(* PLC project PLC, Beckhoff Automation GmbH TwinCAT PLC Control 3.5.21.60 *)
(* stored: creationDateTime 2026-08-05T00:25:24.1454129, modificationDateTime 2026-08-05T00:25:24.1454129 *)

FUNCTION FC_ConcatAll : STRING
VAR_INPUT
	asConcattables					:	ARRAY[0..100] OF STRING;
END_VAR
VAR
	i								:	INT;
	sActual							:	STRING;
	//bStart							:	BOOL := TRUE;
END_VAR

            FOR i := 0 TO 100 BY 1 DO
	IF asConcattables[i] <> '' THEN
		sActual := CONCAT(STR1 := sActual , STR2 := asConcattables[i]);
	END_IF
END_FOR

FC_ConcatAll := sActual;

          
END_FUNCTION

FUNCTION FUN_Build_String_5 : String(255)
VAR_INPUT
	sString_1			:STRING(255);
	sString_2			:STRING(255);
	sString_3			:STRING(255);
	sString_4			:STRING(255);
	sString_5			:STRING(255);
END_VAR
VAR
END_VAR

            IF sString_1 <> ''
	AND sString_2 <>'' 	AND sString_3 <>'' 	AND sString_4 <>'' 	AND sString_5 <>'' THEN
	
	FUN_Build_String_5:=concat(sString_1,concat(sString_2,concat(sString_3,concat(sString_4,sString_5))));
	
ELSIF sString_1 <> ''
	AND sString_2 <>'' 	AND sString_3 <>'' 	AND sString_4 <>'' THEN
	
	FUN_Build_String_5:=concat(sString_1,concat(sString_2,concat(sString_3,sString_4)));
ELSIF sString_1 <> ''
	AND sString_2 <>'' 	AND sString_3 <>'' THEN
	
	FUN_Build_String_5:=concat(sString_1,concat(sString_2,sString_3));
ELSIF sString_1 <> ''AND sString_2 <>'' THEN
	
	FUN_Build_String_5:=concat(sString_1,sString_2);
ELSE
	FUN_Build_String_5:='';
END_IF
          
END_FUNCTION

FUNCTION FUN_Build_String_10 : String(255)
VAR_INPUT
	sString_1			:STRING(255);
	sString_2			:STRING(255);
	sString_3			:STRING(255);
	sString_4			:STRING(255);
	sString_5			:STRING(255);
	sString_6			:STRING(255);
	sString_7			:STRING(255);
	sString_8			:STRING(255);
	sString_9			:STRING(255);
	sString_10			:STRING(255);
END_VAR
VAR
END_VAR

            IF sString_1 <> ''
	AND sString_2 <>'' 	AND sString_3 <>'' 	AND sString_4 <>'' 	AND sString_5 <>'' 	AND sString_6 <>''	AND sString_7 <>''	AND sString_8 <>''
	AND sString_9 <>''	AND sString_10 <>''	 THEN
	
	FUN_Build_String_10:=concat(sString_1,concat(sString_2,concat(sString_3,concat(sString_4,concat
					(sString_5,concat(sString_6,concat(sString_7,concat(sString_8,concat(sString_9,sString_10)))))))));	
ELSIF sString_1 <> ''
	AND sString_2 <>'' 	AND sString_3 <>'' 	AND sString_4 <>'' 	AND sString_5 <>'' 	AND sString_6 <>''	AND sString_7 <>''	AND sString_8 <>''
	AND sString_9 <>'' THEN
	
	FUN_Build_String_10:=concat(sString_1,concat(sString_2,concat(sString_3,concat(sString_4,concat
					(sString_5,concat(sString_6,concat(sString_7,concat(sString_8,sString_9))))))));	
ELSIF sString_1 <> ''
	AND sString_2 <>'' 	AND sString_3 <>'' 	AND sString_4 <>'' 	AND sString_5 <>'' 	AND sString_6 <>''	AND sString_7 <>''	AND sString_8 <>'' THEN
	
	FUN_Build_String_10:=concat(sString_1,concat(sString_2,concat(sString_3,concat(sString_4,concat
					(sString_5,concat(sString_6,concat(sString_7,sString_8)))))));
ELSIF sString_1 <> ''
	AND sString_2 <>'' 	AND sString_3 <>'' 	AND sString_4 <>'' 	AND sString_5 <>'' 	AND sString_6 <>''	AND sString_7 <>'' THEN
	
	FUN_Build_String_10:=concat(sString_1,concat(sString_2,concat(sString_3,concat(sString_4,concat
					(sString_5,concat(sString_6,sString_7))))));
ELSIF sString_1 <> ''
	AND sString_2 <>'' 	AND sString_3 <>'' 	AND sString_4 <>'' 	AND sString_5 <>'' 	AND sString_6 <>'' THEN
	
	FUN_Build_String_10:=concat(sString_1,concat(sString_2,concat(sString_3,concat(sString_4,concat
					(sString_5,sString_6)))));
ELSIF sString_1 <> ''
	AND sString_2 <>'' 	AND sString_3 <>'' 	AND sString_4 <>'' 	AND sString_5 <>'' THEN
	
	FUN_Build_String_10:=concat(sString_1,concat(sString_2,concat(sString_3,concat(sString_4,sString_5))));
	
ELSIF sString_1 <> ''
	AND sString_2 <>'' 	AND sString_3 <>'' 	AND sString_4 <>'' THEN
	
	FUN_Build_String_10:=concat(sString_1,concat(sString_2,concat(sString_3,sString_4)));
ELSIF sString_1 <> ''
	AND sString_2 <>'' 	AND sString_3 <>'' THEN
	
	FUN_Build_String_10:=concat(sString_1,concat(sString_2,sString_3));
ELSIF sString_1 <> ''AND sString_2 <>'' THEN
	
	FUN_Build_String_10:=concat(sString_1,sString_2);
ELSE
	FUN_Build_String_10:='';
END_IF
          
END_FUNCTION

FUNCTION FUN_Build_String_20 : String(255)
VAR_INPUT
	sString_1			:STRING(255);
	sString_2			:STRING(255);
	sString_3			:STRING(255);
	sString_4			:STRING(255);
	sString_5			:STRING(255);
	sString_6			:STRING(255);
	sString_7			:STRING(255);
	sString_8			:STRING(255);
	sString_9			:STRING(255);
	sString_10			:STRING(255);
	sString_11			:STRING(255);
	sString_12			:STRING(255);
	sString_13			:STRING(255);
	sString_14			:STRING(255);
	sString_15			:STRING(255);
	sString_16			:STRING(255);
	sString_17			:STRING(255);
	sString_18			:STRING(255);
	sString_19			:STRING(255);
	sString_20			:STRING(255);
END_VAR
VAR
END_VAR

            IF sString_1 <> ''
	AND sString_2 <>'' 	AND sString_3 <>'' 	AND sString_4 <>'' 	AND sString_5 <>'' 	AND sString_6 <>''	AND sString_7 <>''	AND sString_8 <>''
	AND sString_9 <>''	AND sString_10 <>''	AND sString_11 <>''	AND sString_12 <>'' AND sString_13 <>''	AND sString_14 <>''	AND sString_15 <>''
	AND sString_16 <>''	AND sString_17 <>''	AND sString_18 <>''	AND sString_19 <>''	AND sString_20 <>'' THEN
	
	FUN_Build_String_20:=concat(sString_1,concat(sString_2,concat(sString_3,concat(sString_4,concat
					(sString_5,concat(sString_6,concat(sString_7,concat(sString_8,concat(sString_9,
						concat(sString_10,concat(sString_11,concat(sString_12,concat(sString_13,concat(sString_14,
							concat(sString_15,concat(sString_16,concat(sString_17,concat(sString_18,concat(sString_19,sString_20)))))))))))))))))));
ELSIF sString_1 <> ''
	AND sString_2 <>'' 	AND sString_3 <>'' 	AND sString_4 <>'' 	AND sString_5 <>'' 	AND sString_6 <>''	AND sString_7 <>''	AND sString_8 <>''
	AND sString_9 <>''	AND sString_10 <>''	AND sString_11 <>''	AND sString_12 <>'' AND sString_13 <>''	AND sString_14 <>''	AND sString_15 <>''
	AND sString_16 <>''	AND sString_17 <>''	AND sString_18 <>''	AND sString_19 <>''	 THEN
	
	FUN_Build_String_20:=concat(sString_1,concat(sString_2,concat(sString_3,concat(sString_4,concat
					(sString_5,concat(sString_6,concat(sString_7,concat(sString_8,concat(sString_9,
						concat(sString_10,concat(sString_11,concat(sString_12,concat(sString_13,concat(sString_14,
							concat(sString_15,concat(sString_16,concat(sString_17,concat(sString_18,sString_19))))))))))))))))));
ELSIF sString_1 <> ''
	AND sString_2 <>'' 	AND sString_3 <>'' 	AND sString_4 <>'' 	AND sString_5 <>'' 	AND sString_6 <>''	AND sString_7 <>''	AND sString_8 <>''
	AND sString_9 <>''	AND sString_10 <>''	AND sString_11 <>''	AND sString_12 <>'' AND sString_13 <>''	AND sString_14 <>''	AND sString_15 <>''
	AND sString_16 <>''	AND sString_17 <>''	AND sString_18 <>'' THEN
	
	FUN_Build_String_20:=concat(sString_1,concat(sString_2,concat(sString_3,concat(sString_4,concat
					(sString_5,concat(sString_6,concat(sString_7,concat(sString_8,concat(sString_9,
						concat(sString_10,concat(sString_11,concat(sString_12,concat(sString_13,concat(sString_14,
							concat(sString_15,concat(sString_16,concat(sString_17,sString_18)))))))))))))))));	
ELSIF sString_1 <> ''
	AND sString_2 <>'' 	AND sString_3 <>'' 	AND sString_4 <>'' 	AND sString_5 <>'' 	AND sString_6 <>''	AND sString_7 <>''	AND sString_8 <>''
	AND sString_9 <>''	AND sString_10 <>''	AND sString_11 <>''	AND sString_12 <>'' AND sString_13 <>''	AND sString_14 <>''	AND sString_15 <>''
	AND sString_16 <>''	AND sString_17 <>'' THEN
	
	FUN_Build_String_20:=concat(sString_1,concat(sString_2,concat(sString_3,concat(sString_4,concat
					(sString_5,concat(sString_6,concat(sString_7,concat(sString_8,concat(sString_9,
						concat(sString_10,concat(sString_11,concat(sString_12,concat(sString_13,concat(sString_14,
							concat(sString_15,concat(sString_16,sString_17))))))))))))))));	
ELSIF sString_1 <> ''
	AND sString_2 <>'' 	AND sString_3 <>'' 	AND sString_4 <>'' 	AND sString_5 <>'' 	AND sString_6 <>''	AND sString_7 <>''	AND sString_8 <>''
	AND sString_9 <>''	AND sString_10 <>''	AND sString_11 <>''	AND sString_12 <>'' AND sString_13 <>''	AND sString_14 <>''	AND sString_15 <>''
	AND sString_16 <>''	THEN
	
	FUN_Build_String_20:=concat(sString_1,concat(sString_2,concat(sString_3,concat(sString_4,concat
					(sString_5,concat(sString_6,concat(sString_7,concat(sString_8,concat(sString_9,
						concat(sString_10,concat(sString_11,concat(sString_12,concat(sString_13,concat(sString_14,
							concat(sString_15,sString_16)))))))))))))));	
ELSIF sString_1 <> ''
	AND sString_2 <>'' 	AND sString_3 <>'' 	AND sString_4 <>'' 	AND sString_5 <>'' 	AND sString_6 <>''	AND sString_7 <>''	AND sString_8 <>''
	AND sString_9 <>''	AND sString_10 <>''	AND sString_11 <>''	AND sString_12 <>'' AND sString_13 <>''	AND sString_14 <>''	AND sString_15 <>''	THEN
	
	FUN_Build_String_20:=concat(sString_1,concat(sString_2,concat(sString_3,concat(sString_4,concat
					(sString_5,concat(sString_6,concat(sString_7,concat(sString_8,concat(sString_9,
						concat(sString_10,concat(sString_11,concat(sString_12,concat(sString_13,concat(sString_14,sString_15))))))))))))));	
ELSIF sString_1 <> ''
	AND sString_2 <>'' 	AND sString_3 <>'' 	AND sString_4 <>'' 	AND sString_5 <>'' 	AND sString_6 <>''	AND sString_7 <>''	AND sString_8 <>''
	AND sString_9 <>''	AND sString_10 <>''	AND sString_11 <>''	AND sString_12 <>'' AND sString_13 <>''	AND sString_14 <>'' THEN
	
	FUN_Build_String_20:=concat(sString_1,concat(sString_2,concat(sString_3,concat(sString_4,concat
					(sString_5,concat(sString_6,concat(sString_7,concat(sString_8,concat(sString_9,
						concat(sString_10,concat(sString_11,concat(sString_12,concat(sString_13,sString_14)))))))))))));	
ELSIF sString_1 <> ''
	AND sString_2 <>'' 	AND sString_3 <>'' 	AND sString_4 <>'' 	AND sString_5 <>'' 	AND sString_6 <>''	AND sString_7 <>''	AND sString_8 <>''
	AND sString_9 <>''	AND sString_10 <>''	AND sString_11 <>''	AND sString_12 <>'' AND sString_13 <>'' THEN
	
	FUN_Build_String_20:=concat(sString_1,concat(sString_2,concat(sString_3,concat(sString_4,concat
					(sString_5,concat(sString_6,concat(sString_7,concat(sString_8,concat(sString_9,
						concat(sString_10,concat(sString_11,concat(sString_12,sString_13))))))))))));	
ELSIF sString_1 <> ''
	AND sString_2 <>'' 	AND sString_3 <>'' 	AND sString_4 <>'' 	AND sString_5 <>'' 	AND sString_6 <>''	AND sString_7 <>''	AND sString_8 <>''
	AND sString_9 <>''	AND sString_10 <>''	AND sString_11 <>''	AND sString_12 <>'' THEN
	
	FUN_Build_String_20:=concat(sString_1,concat(sString_2,concat(sString_3,concat(sString_4,concat
					(sString_5,concat(sString_6,concat(sString_7,concat(sString_8,concat(sString_9,
						concat(sString_10,concat(sString_11,sString_12)))))))))));	
ELSIF sString_1 <> ''
	AND sString_2 <>'' 	AND sString_3 <>'' 	AND sString_4 <>'' 	AND sString_5 <>'' 	AND sString_6 <>''	AND sString_7 <>''	AND sString_8 <>''
	AND sString_9 <>''	AND sString_10 <>''	AND sString_11 <>'' THEN
	
	FUN_Build_String_20:=concat(sString_1,concat(sString_2,concat(sString_3,concat(sString_4,concat
					(sString_5,concat(sString_6,concat(sString_7,concat(sString_8,concat(sString_9,
						concat(sString_10,sString_11))))))))));	
ELSIF sString_1 <> ''
	AND sString_2 <>'' 	AND sString_3 <>'' 	AND sString_4 <>'' 	AND sString_5 <>'' 	AND sString_6 <>''	AND sString_7 <>''	AND sString_8 <>''
	AND sString_9 <>''	AND sString_10 <>''	 THEN
	
	FUN_Build_String_20:=concat(sString_1,concat(sString_2,concat(sString_3,concat(sString_4,concat
					(sString_5,concat(sString_6,concat(sString_7,concat(sString_8,concat(sString_9,sString_10)))))))));	
ELSIF sString_1 <> ''
	AND sString_2 <>'' 	AND sString_3 <>'' 	AND sString_4 <>'' 	AND sString_5 <>'' 	AND sString_6 <>''	AND sString_7 <>''	AND sString_8 <>''
	AND sString_9 <>'' THEN
	
	FUN_Build_String_20:=concat(sString_1,concat(sString_2,concat(sString_3,concat(sString_4,concat
					(sString_5,concat(sString_6,concat(sString_7,concat(sString_8,sString_9))))))));	
ELSIF sString_1 <> ''
	AND sString_2 <>'' 	AND sString_3 <>'' 	AND sString_4 <>'' 	AND sString_5 <>'' 	AND sString_6 <>''	AND sString_7 <>''	AND sString_8 <>'' THEN
	
	FUN_Build_String_20:=concat(sString_1,concat(sString_2,concat(sString_3,concat(sString_4,concat
					(sString_5,concat(sString_6,concat(sString_7,sString_8)))))));
ELSIF sString_1 <> ''
	AND sString_2 <>'' 	AND sString_3 <>'' 	AND sString_4 <>'' 	AND sString_5 <>'' 	AND sString_6 <>''	AND sString_7 <>'' THEN
	
	FUN_Build_String_20:=concat(sString_1,concat(sString_2,concat(sString_3,concat(sString_4,concat
					(sString_5,concat(sString_6,sString_7))))));
ELSIF sString_1 <> ''
	AND sString_2 <>'' 	AND sString_3 <>'' 	AND sString_4 <>'' 	AND sString_5 <>'' 	AND sString_6 <>'' THEN
	
	FUN_Build_String_20:=concat(sString_1,concat(sString_2,concat(sString_3,concat(sString_4,concat
					(sString_5,sString_6)))));
ELSIF sString_1 <> ''
	AND sString_2 <>'' 	AND sString_3 <>'' 	AND sString_4 <>'' 	AND sString_5 <>'' THEN
	
	FUN_Build_String_20:=concat(sString_1,concat(sString_2,concat(sString_3,concat(sString_4,sString_5))));
	
ELSIF sString_1 <> ''
	AND sString_2 <>'' 	AND sString_3 <>'' 	AND sString_4 <>'' THEN
	
	FUN_Build_String_20:=concat(sString_1,concat(sString_2,concat(sString_3,sString_4)));
ELSIF sString_1 <> ''
	AND sString_2 <>'' 	AND sString_3 <>'' THEN
	
	FUN_Build_String_20:=concat(sString_1,concat(sString_2,sString_3));
ELSIF sString_1 <> ''AND sString_2 <>'' THEN
	
	FUN_Build_String_20:=concat(sString_1,sString_2);
ELSE
	FUN_Build_String_20:='';
END_IF
          
END_FUNCTION

FUNCTION FUN_Build_String_30 : String(500)
VAR_INPUT
	sString_1			:STRING(255);
	sString_2			:STRING(255);
	sString_3			:STRING(255);
	sString_4			:STRING(255);
	sString_5			:STRING(255);
	sString_6			:STRING(255);
	sString_7			:STRING(255);
	sString_8			:STRING(255);
	sString_9			:STRING(255);
	sString_10			:STRING(255);
	sString_11			:STRING(255);
	sString_12			:STRING(255);
	sString_13			:STRING(255);
	sString_14			:STRING(255);
	sString_15			:STRING(255);
	sString_16			:STRING(255);
	sString_17			:STRING(255);
	sString_18			:STRING(255);
	sString_19			:STRING(255);
	sString_20			:STRING(255);
	sString_21			:STRING(255);
	sString_22			:STRING(255);
	sString_23			:STRING(255);
	sString_24			:STRING(255);
	sString_25			:STRING(255);
	sString_26			:STRING(255);
	sString_27			:STRING(255);
	sString_28			:STRING(255);
	sString_29			:STRING(255);
	sString_30			:STRING(255);
END_VAR
VAR
END_VAR

            IF sString_1 <> ''
	AND sString_2 <>'' 	AND sString_3 <>'' 	AND sString_4 <>'' 	AND sString_5 <>'' 	AND sString_6 <>''	AND sString_7 <>''	AND sString_8 <>''
	AND sString_9 <>''	AND sString_10 <>''	AND sString_11 <>''	AND sString_12 <>'' AND sString_13 <>''	AND sString_14 <>''	AND sString_15 <>''
	AND sString_16 <>''	AND sString_17 <>''	AND sString_18 <>''	AND sString_19 <>''	AND sString_20 <>'' AND sString_21 <>'' AND sString_22 <>''
	AND sString_23 <>'' AND sString_24 <>'' AND sString_25 <>'' AND sString_26 <>'' AND sString_27 <>'' AND sString_28 <>'' AND sString_29 <>'' 
	AND sString_30 <>''THEN
	
	FUN_Build_String_30:=concat(sString_1,concat(sString_2,concat(sString_3,concat(sString_4,concat
					(sString_5,concat(sString_6,concat(sString_7,concat(sString_8,concat(sString_9,
						concat(sString_10,concat(sString_11,concat(sString_12,concat(sString_13,concat(sString_14,
							concat(sString_15,concat(sString_16,concat(sString_17,concat(sString_18,concat(sString_19,concat(sString_20,
								concat(sString_21,concat(sString_22,concat(sString_23,concat(sString_24,concat(sString_25,concat(sString_26,
									concat(sString_27,concat(sString_28,concat(sString_29,sString_30)))))))))))))))))))))))))))));

ELSIF sString_1 <> ''
	AND sString_2 <>'' 	AND sString_3 <>'' 	AND sString_4 <>'' 	AND sString_5 <>'' 	AND sString_6 <>''	AND sString_7 <>''	AND sString_8 <>''
	AND sString_9 <>''	AND sString_10 <>''	AND sString_11 <>''	AND sString_12 <>'' AND sString_13 <>''	AND sString_14 <>''	AND sString_15 <>''
	AND sString_16 <>''	AND sString_17 <>''	AND sString_18 <>''	AND sString_19 <>''	AND sString_20 <>'' AND sString_21 <>'' AND sString_22 <>''
	AND sString_23 <>'' AND sString_24 <>'' AND sString_25 <>'' AND sString_26 <>'' AND sString_27 <>'' AND sString_28 <>'' AND sString_29 <>''THEN
	
	FUN_Build_String_30:=concat(sString_1,concat(sString_2,concat(sString_3,concat(sString_4,concat
					(sString_5,concat(sString_6,concat(sString_7,concat(sString_8,concat(sString_9,
						concat(sString_10,concat(sString_11,concat(sString_12,concat(sString_13,concat(sString_14,
							concat(sString_15,concat(sString_16,concat(sString_17,concat(sString_18,concat(sString_19,concat(sString_20,
								concat(sString_21,concat(sString_22,concat(sString_23,concat(sString_24,concat(sString_25,concat(sString_26,
									concat(sString_27,concat(sString_28,sString_29))))))))))))))))))))))))))));
ELSIF sString_1 <> ''
	AND sString_2 <>'' 	AND sString_3 <>'' 	AND sString_4 <>'' 	AND sString_5 <>'' 	AND sString_6 <>''	AND sString_7 <>''	AND sString_8 <>''
	AND sString_9 <>''	AND sString_10 <>''	AND sString_11 <>''	AND sString_12 <>'' AND sString_13 <>''	AND sString_14 <>''	AND sString_15 <>''
	AND sString_16 <>''	AND sString_17 <>''	AND sString_18 <>''	AND sString_19 <>''	AND sString_20 <>'' AND sString_21 <>'' AND sString_22 <>''
	AND sString_23 <>'' AND sString_24 <>'' AND sString_25 <>'' AND sString_26 <>'' AND sString_27 <>'' AND sString_28 <>''THEN
	
	FUN_Build_String_30:=concat(sString_1,concat(sString_2,concat(sString_3,concat(sString_4,concat
					(sString_5,concat(sString_6,concat(sString_7,concat(sString_8,concat(sString_9,
						concat(sString_10,concat(sString_11,concat(sString_12,concat(sString_13,concat(sString_14,
							concat(sString_15,concat(sString_16,concat(sString_17,concat(sString_18,concat(sString_19,concat(sString_20,
								concat(sString_21,concat(sString_22,concat(sString_23,concat(sString_24,concat(sString_25,concat(sString_26,
									concat(sString_27,sString_28)))))))))))))))))))))))))));
ELSIF sString_1 <> ''
	AND sString_2 <>'' 	AND sString_3 <>'' 	AND sString_4 <>'' 	AND sString_5 <>'' 	AND sString_6 <>''	AND sString_7 <>''	AND sString_8 <>''
	AND sString_9 <>''	AND sString_10 <>''	AND sString_11 <>''	AND sString_12 <>'' AND sString_13 <>''	AND sString_14 <>''	AND sString_15 <>''
	AND sString_16 <>''	AND sString_17 <>''	AND sString_18 <>''	AND sString_19 <>''	AND sString_20 <>'' AND sString_21 <>'' AND sString_22 <>''
	AND sString_23 <>'' AND sString_24 <>'' AND sString_25 <>'' AND sString_26 <>'' AND sString_27 <>''THEN
	
	FUN_Build_String_30:=concat(sString_1,concat(sString_2,concat(sString_3,concat(sString_4,concat
					(sString_5,concat(sString_6,concat(sString_7,concat(sString_8,concat(sString_9,
						concat(sString_10,concat(sString_11,concat(sString_12,concat(sString_13,concat(sString_14,
							concat(sString_15,concat(sString_16,concat(sString_17,concat(sString_18,concat(sString_19,concat(sString_20,
								concat(sString_21,concat(sString_22,concat(sString_23,concat(sString_24,concat(sString_25,concat(sString_26,sString_27))))))))))))))))))))))))));

ELSIF sString_1 <> ''
	AND sString_2 <>'' 	AND sString_3 <>'' 	AND sString_4 <>'' 	AND sString_5 <>'' 	AND sString_6 <>''	AND sString_7 <>''	AND sString_8 <>''
	AND sString_9 <>''	AND sString_10 <>''	AND sString_11 <>''	AND sString_12 <>'' AND sString_13 <>''	AND sString_14 <>''	AND sString_15 <>''
	AND sString_16 <>''	AND sString_17 <>''	AND sString_18 <>''	AND sString_19 <>''	AND sString_20 <>'' AND sString_21 <>'' AND sString_22 <>''
	AND sString_23 <>'' AND sString_24 <>'' AND sString_25 <>'' AND sString_26 <>''THEN
	
	FUN_Build_String_30:=concat(sString_1,concat(sString_2,concat(sString_3,concat(sString_4,concat
					(sString_5,concat(sString_6,concat(sString_7,concat(sString_8,concat(sString_9,
						concat(sString_10,concat(sString_11,concat(sString_12,concat(sString_13,concat(sString_14,
							concat(sString_15,concat(sString_16,concat(sString_17,concat(sString_18,concat(sString_19,concat(sString_20,
								concat(sString_21,concat(sString_22,concat(sString_23,concat(sString_24,concat(sString_25,sString_26)))))))))))))))))))))))));
ELSIF sString_1 <> ''
	AND sString_2 <>'' 	AND sString_3 <>'' 	AND sString_4 <>'' 	AND sString_5 <>'' 	AND sString_6 <>''	AND sString_7 <>''	AND sString_8 <>''
	AND sString_9 <>''	AND sString_10 <>''	AND sString_11 <>''	AND sString_12 <>'' AND sString_13 <>''	AND sString_14 <>''	AND sString_15 <>''
	AND sString_16 <>''	AND sString_17 <>''	AND sString_18 <>''	AND sString_19 <>''	AND sString_20 <>'' AND sString_21 <>'' AND sString_22 <>''
	AND sString_23 <>'' AND sString_24 <>'' AND sString_25 <>''THEN
	
	FUN_Build_String_30:=concat(sString_1,concat(sString_2,concat(sString_3,concat(sString_4,concat
					(sString_5,concat(sString_6,concat(sString_7,concat(sString_8,concat(sString_9,
						concat(sString_10,concat(sString_11,concat(sString_12,concat(sString_13,concat(sString_14,
							concat(sString_15,concat(sString_16,concat(sString_17,concat(sString_18,concat(sString_19,concat(sString_20,
								concat(sString_21,concat(sString_22,concat(sString_23,concat(sString_24,sString_25))))))))))))))))))))))));
ELSIF sString_1 <> ''
	AND sString_2 <>'' 	AND sString_3 <>'' 	AND sString_4 <>'' 	AND sString_5 <>'' 	AND sString_6 <>''	AND sString_7 <>''	AND sString_8 <>''
	AND sString_9 <>''	AND sString_10 <>''	AND sString_11 <>''	AND sString_12 <>'' AND sString_13 <>''	AND sString_14 <>''	AND sString_15 <>''
	AND sString_16 <>''	AND sString_17 <>''	AND sString_18 <>''	AND sString_19 <>''	AND sString_20 <>'' AND sString_21 <>'' AND sString_22 <>''
	AND sString_23 <>'' AND sString_24 <>''THEN
	
	FUN_Build_String_30:=concat(sString_1,concat(sString_2,concat(sString_3,concat(sString_4,concat
					(sString_5,concat(sString_6,concat(sString_7,concat(sString_8,concat(sString_9,
						concat(sString_10,concat(sString_11,concat(sString_12,concat(sString_13,concat(sString_14,
							concat(sString_15,concat(sString_16,concat(sString_17,concat(sString_18,concat(sString_19,concat(sString_20,
								concat(sString_21,concat(sString_22,concat(sString_23,sString_24)))))))))))))))))))))));
ELSIF sString_1 <> ''
	AND sString_2 <>'' 	AND sString_3 <>'' 	AND sString_4 <>'' 	AND sString_5 <>'' 	AND sString_6 <>''	AND sString_7 <>''	AND sString_8 <>''
	AND sString_9 <>''	AND sString_10 <>''	AND sString_11 <>''	AND sString_12 <>'' AND sString_13 <>''	AND sString_14 <>''	AND sString_15 <>''
	AND sString_16 <>''	AND sString_17 <>''	AND sString_18 <>''	AND sString_19 <>''	AND sString_20 <>'' AND sString_21 <>'' AND sString_22 <>''
	AND sString_23 <>''THEN
	
	FUN_Build_String_30:=concat(sString_1,concat(sString_2,concat(sString_3,concat(sString_4,concat
					(sString_5,concat(sString_6,concat(sString_7,concat(sString_8,concat(sString_9,
						concat(sString_10,concat(sString_11,concat(sString_12,concat(sString_13,concat(sString_14,
							concat(sString_15,concat(sString_16,concat(sString_17,concat(sString_18,concat(sString_19,concat(sString_20,
								concat(sString_21,concat(sString_22,sString_23))))))))))))))))))))));
ELSIF sString_1 <> ''
	AND sString_2 <>'' 	AND sString_3 <>'' 	AND sString_4 <>'' 	AND sString_5 <>'' 	AND sString_6 <>''	AND sString_7 <>''	AND sString_8 <>''
	AND sString_9 <>''	AND sString_10 <>''	AND sString_11 <>''	AND sString_12 <>'' AND sString_13 <>''	AND sString_14 <>''	AND sString_15 <>''
	AND sString_16 <>''	AND sString_17 <>''	AND sString_18 <>''	AND sString_19 <>''	AND sString_20 <>'' AND sString_21 <>'' AND sString_22 <>''THEN
	
	FUN_Build_String_30:=concat(sString_1,concat(sString_2,concat(sString_3,concat(sString_4,concat
					(sString_5,concat(sString_6,concat(sString_7,concat(sString_8,concat(sString_9,
						concat(sString_10,concat(sString_11,concat(sString_12,concat(sString_13,concat(sString_14,
							concat(sString_15,concat(sString_16,concat(sString_17,concat(sString_18,concat(sString_19,concat(sString_20,concat(sString_21,sString_22)))))))))))))))))))));
ELSIF sString_1 <> ''
	AND sString_2 <>'' 	AND sString_3 <>'' 	AND sString_4 <>'' 	AND sString_5 <>'' 	AND sString_6 <>''	AND sString_7 <>''	AND sString_8 <>''
	AND sString_9 <>''	AND sString_10 <>''	AND sString_11 <>''	AND sString_12 <>'' AND sString_13 <>''	AND sString_14 <>''	AND sString_15 <>''
	AND sString_16 <>''	AND sString_17 <>''	AND sString_18 <>''	AND sString_19 <>''	AND sString_20 <>'' AND sString_21 <>''THEN
	
	FUN_Build_String_30:=concat(sString_1,concat(sString_2,concat(sString_3,concat(sString_4,concat
					(sString_5,concat(sString_6,concat(sString_7,concat(sString_8,concat(sString_9,
						concat(sString_10,concat(sString_11,concat(sString_12,concat(sString_13,concat(sString_14,
							concat(sString_15,concat(sString_16,concat(sString_17,concat(sString_18,concat(sString_19,concat(sString_20,sString_21))))))))))))))))))));
ELSIF sString_1 <> ''
	AND sString_2 <>'' 	AND sString_3 <>'' 	AND sString_4 <>'' 	AND sString_5 <>'' 	AND sString_6 <>''	AND sString_7 <>''	AND sString_8 <>''
	AND sString_9 <>''	AND sString_10 <>''	AND sString_11 <>''	AND sString_12 <>'' AND sString_13 <>''	AND sString_14 <>''	AND sString_15 <>''
	AND sString_16 <>''	AND sString_17 <>''	AND sString_18 <>''	AND sString_19 <>''	AND sString_20 <>'' THEN
	
	FUN_Build_String_30:=concat(sString_1,concat(sString_2,concat(sString_3,concat(sString_4,concat
					(sString_5,concat(sString_6,concat(sString_7,concat(sString_8,concat(sString_9,
						concat(sString_10,concat(sString_11,concat(sString_12,concat(sString_13,concat(sString_14,
							concat(sString_15,concat(sString_16,concat(sString_17,concat(sString_18,concat(sString_19,sString_20)))))))))))))))))));
ELSIF sString_1 <> ''
	AND sString_2 <>'' 	AND sString_3 <>'' 	AND sString_4 <>'' 	AND sString_5 <>'' 	AND sString_6 <>''	AND sString_7 <>''	AND sString_8 <>''
	AND sString_9 <>''	AND sString_10 <>''	AND sString_11 <>''	AND sString_12 <>'' AND sString_13 <>''	AND sString_14 <>''	AND sString_15 <>''
	AND sString_16 <>''	AND sString_17 <>''	AND sString_18 <>''	AND sString_19 <>''	 THEN
	
	FUN_Build_String_30:=concat(sString_1,concat(sString_2,concat(sString_3,concat(sString_4,concat
					(sString_5,concat(sString_6,concat(sString_7,concat(sString_8,concat(sString_9,
						concat(sString_10,concat(sString_11,concat(sString_12,concat(sString_13,concat(sString_14,
							concat(sString_15,concat(sString_16,concat(sString_17,concat(sString_18,sString_19))))))))))))))))));
ELSIF sString_1 <> ''
	AND sString_2 <>'' 	AND sString_3 <>'' 	AND sString_4 <>'' 	AND sString_5 <>'' 	AND sString_6 <>''	AND sString_7 <>''	AND sString_8 <>''
	AND sString_9 <>''	AND sString_10 <>''	AND sString_11 <>''	AND sString_12 <>'' AND sString_13 <>''	AND sString_14 <>''	AND sString_15 <>''
	AND sString_16 <>''	AND sString_17 <>''	AND sString_18 <>'' THEN
	
	FUN_Build_String_30:=concat(sString_1,concat(sString_2,concat(sString_3,concat(sString_4,concat
					(sString_5,concat(sString_6,concat(sString_7,concat(sString_8,concat(sString_9,
						concat(sString_10,concat(sString_11,concat(sString_12,concat(sString_13,concat(sString_14,
							concat(sString_15,concat(sString_16,concat(sString_17,sString_18)))))))))))))))));	
ELSIF sString_1 <> ''
	AND sString_2 <>'' 	AND sString_3 <>'' 	AND sString_4 <>'' 	AND sString_5 <>'' 	AND sString_6 <>''	AND sString_7 <>''	AND sString_8 <>''
	AND sString_9 <>''	AND sString_10 <>''	AND sString_11 <>''	AND sString_12 <>'' AND sString_13 <>''	AND sString_14 <>''	AND sString_15 <>''
	AND sString_16 <>''	AND sString_17 <>'' THEN
	
	FUN_Build_String_30:=concat(sString_1,concat(sString_2,concat(sString_3,concat(sString_4,concat
					(sString_5,concat(sString_6,concat(sString_7,concat(sString_8,concat(sString_9,
						concat(sString_10,concat(sString_11,concat(sString_12,concat(sString_13,concat(sString_14,
							concat(sString_15,concat(sString_16,sString_17))))))))))))))));	
ELSIF sString_1 <> ''
	AND sString_2 <>'' 	AND sString_3 <>'' 	AND sString_4 <>'' 	AND sString_5 <>'' 	AND sString_6 <>''	AND sString_7 <>''	AND sString_8 <>''
	AND sString_9 <>''	AND sString_10 <>''	AND sString_11 <>''	AND sString_12 <>'' AND sString_13 <>''	AND sString_14 <>''	AND sString_15 <>''
	AND sString_16 <>''	THEN
	
	FUN_Build_String_30:=concat(sString_1,concat(sString_2,concat(sString_3,concat(sString_4,concat
					(sString_5,concat(sString_6,concat(sString_7,concat(sString_8,concat(sString_9,
						concat(sString_10,concat(sString_11,concat(sString_12,concat(sString_13,concat(sString_14,
							concat(sString_15,sString_16)))))))))))))));	
ELSIF sString_1 <> ''
	AND sString_2 <>'' 	AND sString_3 <>'' 	AND sString_4 <>'' 	AND sString_5 <>'' 	AND sString_6 <>''	AND sString_7 <>''	AND sString_8 <>''
	AND sString_9 <>''	AND sString_10 <>''	AND sString_11 <>''	AND sString_12 <>'' AND sString_13 <>''	AND sString_14 <>''	AND sString_15 <>''	THEN
	
	FUN_Build_String_30:=concat(sString_1,concat(sString_2,concat(sString_3,concat(sString_4,concat
					(sString_5,concat(sString_6,concat(sString_7,concat(sString_8,concat(sString_9,
						concat(sString_10,concat(sString_11,concat(sString_12,concat(sString_13,concat(sString_14,sString_15))))))))))))));	
ELSIF sString_1 <> ''
	AND sString_2 <>'' 	AND sString_3 <>'' 	AND sString_4 <>'' 	AND sString_5 <>'' 	AND sString_6 <>''	AND sString_7 <>''	AND sString_8 <>''
	AND sString_9 <>''	AND sString_10 <>''	AND sString_11 <>''	AND sString_12 <>'' AND sString_13 <>''	AND sString_14 <>'' THEN
	
	FUN_Build_String_30:=concat(sString_1,concat(sString_2,concat(sString_3,concat(sString_4,concat
					(sString_5,concat(sString_6,concat(sString_7,concat(sString_8,concat(sString_9,
						concat(sString_10,concat(sString_11,concat(sString_12,concat(sString_13,sString_14)))))))))))));	
ELSIF sString_1 <> ''
	AND sString_2 <>'' 	AND sString_3 <>'' 	AND sString_4 <>'' 	AND sString_5 <>'' 	AND sString_6 <>''	AND sString_7 <>''	AND sString_8 <>''
	AND sString_9 <>''	AND sString_10 <>''	AND sString_11 <>''	AND sString_12 <>'' AND sString_13 <>'' THEN
	
	FUN_Build_String_30:=concat(sString_1,concat(sString_2,concat(sString_3,concat(sString_4,concat
					(sString_5,concat(sString_6,concat(sString_7,concat(sString_8,concat(sString_9,
						concat(sString_10,concat(sString_11,concat(sString_12,sString_13))))))))))));	
ELSIF sString_1 <> ''
	AND sString_2 <>'' 	AND sString_3 <>'' 	AND sString_4 <>'' 	AND sString_5 <>'' 	AND sString_6 <>''	AND sString_7 <>''	AND sString_8 <>''
	AND sString_9 <>''	AND sString_10 <>''	AND sString_11 <>''	AND sString_12 <>'' THEN
	
	FUN_Build_String_30:=concat(sString_1,concat(sString_2,concat(sString_3,concat(sString_4,concat
					(sString_5,concat(sString_6,concat(sString_7,concat(sString_8,concat(sString_9,
						concat(sString_10,concat(sString_11,sString_12)))))))))));	
ELSIF sString_1 <> ''
	AND sString_2 <>'' 	AND sString_3 <>'' 	AND sString_4 <>'' 	AND sString_5 <>'' 	AND sString_6 <>''	AND sString_7 <>''	AND sString_8 <>''
	AND sString_9 <>''	AND sString_10 <>''	AND sString_11 <>'' THEN
	
	FUN_Build_String_30:=concat(sString_1,concat(sString_2,concat(sString_3,concat(sString_4,concat
					(sString_5,concat(sString_6,concat(sString_7,concat(sString_8,concat(sString_9,
						concat(sString_10,sString_11))))))))));	
ELSIF sString_1 <> ''
	AND sString_2 <>'' 	AND sString_3 <>'' 	AND sString_4 <>'' 	AND sString_5 <>'' 	AND sString_6 <>''	AND sString_7 <>''	AND sString_8 <>''
	AND sString_9 <>''	AND sString_10 <>''	 THEN
	
	FUN_Build_String_30:=concat(sString_1,concat(sString_2,concat(sString_3,concat(sString_4,concat
					(sString_5,concat(sString_6,concat(sString_7,concat(sString_8,concat(sString_9,sString_10)))))))));	
ELSIF sString_1 <> ''
	AND sString_2 <>'' 	AND sString_3 <>'' 	AND sString_4 <>'' 	AND sString_5 <>'' 	AND sString_6 <>''	AND sString_7 <>''	AND sString_8 <>''
	AND sString_9 <>'' THEN
	
	FUN_Build_String_30:=concat(sString_1,concat(sString_2,concat(sString_3,concat(sString_4,concat
					(sString_5,concat(sString_6,concat(sString_7,concat(sString_8,sString_9))))))));	
ELSIF sString_1 <> ''
	AND sString_2 <>'' 	AND sString_3 <>'' 	AND sString_4 <>'' 	AND sString_5 <>'' 	AND sString_6 <>''	AND sString_7 <>''	AND sString_8 <>'' THEN
	
	FUN_Build_String_30:=concat(sString_1,concat(sString_2,concat(sString_3,concat(sString_4,concat
					(sString_5,concat(sString_6,concat(sString_7,sString_8)))))));
ELSIF sString_1 <> ''
	AND sString_2 <>'' 	AND sString_3 <>'' 	AND sString_4 <>'' 	AND sString_5 <>'' 	AND sString_6 <>''	AND sString_7 <>'' THEN
	
	FUN_Build_String_30:=concat(sString_1,concat(sString_2,concat(sString_3,concat(sString_4,concat
					(sString_5,concat(sString_6,sString_7))))));
ELSIF sString_1 <> ''
	AND sString_2 <>'' 	AND sString_3 <>'' 	AND sString_4 <>'' 	AND sString_5 <>'' 	AND sString_6 <>'' THEN
	
	FUN_Build_String_30:=concat(sString_1,concat(sString_2,concat(sString_3,concat(sString_4,concat
					(sString_5,sString_6)))));
ELSIF sString_1 <> ''
	AND sString_2 <>'' 	AND sString_3 <>'' 	AND sString_4 <>'' 	AND sString_5 <>'' THEN
	
	FUN_Build_String_30:=concat(sString_1,concat(sString_2,concat(sString_3,concat(sString_4,sString_5))));
	
ELSIF sString_1 <> ''
	AND sString_2 <>'' 	AND sString_3 <>'' 	AND sString_4 <>'' THEN
	
	FUN_Build_String_30:=concat(sString_1,concat(sString_2,concat(sString_3,sString_4)));
ELSIF sString_1 <> ''
	AND sString_2 <>'' 	AND sString_3 <>'' THEN
	
	FUN_Build_String_30:=concat(sString_1,concat(sString_2,sString_3));
ELSIF sString_1 <> ''AND sString_2 <>'' THEN
	
	FUN_Build_String_30:=concat(sString_1,sString_2);
ELSE
	FUN_Build_String_30:='';
END_IF
          
END_FUNCTION

FUNCTION FUN_Concat_String_100 : STRING [1000]
VAR_INPUT
	arrString:	ARRAY [1..100] OF STRING(1000);
END_VAR
VAR
	i: INT;
	j: INT;
	k: INT;
	iArchive_j		:INT;
	arrTMP255Byte		:ARRAY [1..1000] OF BYTE;
	arrAllStringInByte		:ARRAY [1..1000] OF BYTE;
	sTemp			:STRING(1000);
	iTest1: INT;
	iTest2: UINT;
END_VAR

            //	FUN_Concat_String_100:='ERROR FUN_Concat_String_100 to many input character!!!';
MEMSET(ADR(arrAllStringInByte),STRING_TO_BYTE(''),SIZEOF(arrAllStringInByte));
j:=1;
iArchive_j:=1;
FOR i:=1 TO 100 DO
	IF arrString[i] <> ''
		OR arrString[i+1] <> '' THEN
			MEMCPY(ADR(arrTMP255Byte),ADR(arrString[i]),1000);
			
			k:=1;
			FOR j:=iArchive_j TO (iArchive_j+1000) DO
				IF arrTMP255Byte[k] <> 0 THEN
					arrAllStringInByte[j]:=arrTMP255Byte[k];
					k:=k+1;
				ELSE
					EXIT;
				END_IF
			END_FOR
			iArchive_j:=j;
			IF iArchive_j >=1000 THEN   //ERROR
				FUN_Concat_String_100:='ERROR FUN_Concat_String_100 to many input character!!!';
				EXIT;
			END_IF
	ELSIF i > 1 THEN					//OK
		 MEMCPY(ADR(FUN_Concat_String_100),ADR(arrAllStringInByte),SIZEOF(arrAllStringInByte)); 
		 EXIT;
	ELSIF i = 1 THEN					//ERROR
		FUN_Concat_String_100:='ERROR FUN_Concat_String_100 received no string to the input!!!';
		EXIT;
	ELSE
		EXIT;
	END_IF	
END_FOR

          
END_FUNCTION

FUNCTION FUN_CutString : STRING(255)
VAR_INPUT
	sRawString							:STRING[1000];
	sStringStartIdentifier				:STRING;
	sStringEndIdentifier				:STRING;
	sDataElementSeparator				:STRING;
END_VAR
VAR
	iStringFound						:INT;// 1--> string found 0--> no string
	sCutString							:STRING;
	iTemp: INT;
	sTempString: STRING(1000);
	iTempStringEnd: INT;
	iLenghtOfCompleteString: INT;
	iLenghtofStartIdentifier: INT;
END_VAR

            iTemp:=find(sRawString,concat(sDataElementSeparator,sStringStartIdentifier));
iLenghtOfCompleteString:=len(sRawString);
iLenghtofStartIdentifier:=len(concat(sDataElementSeparator,sStringStartIdentifier));

IF iTemp > 0 THEN
	IF iLenghtofStartIdentifier > 1 THEN
		sTempString:=right(sRawString,(iLenghtOfCompleteString-iTemp-(iLenghtofStartIdentifier-1)));
	ELSE
		sTempString:=right(sRawString,(iLenghtOfCompleteString-iTemp));
	END_IF
	iTempStringEnd:=find(sTempString,sStringEndIdentifier);
	IF iTempStringEnd > 0 THEN
		FUN_CutString:=MID(sTempString,iTempStringEnd-1,1);
	ELSE
		FUN_CutString:='';	
	END_IF
ELSE
	FUN_CutString:='';
END_IF
          
END_FUNCTION

FUNCTION_BLOCK FB_CutString
VAR_INPUT
	sRawString							:STRING[1000];
	sStringStartIdentifier				:STRING;
	sStringEndIdentifier				:STRING;
	sDataElementSeparator				:STRING;
END_VAR
VAR_OUTPUT
	iStringFound						:INT;// 1--> string found 0--> no string
	sCutString							:STRING;
END_VAR
VAR
	iTemp: INT;
	sTempString: STRING(1000);
	iTempStringEnd: INT;
	iLenghtOfCompleteString: INT;
	iLenghtofStartIdentifier: INT;
END_VAR

            iTemp:=find(sRawString,concat(sDataElementSeparator,sStringStartIdentifier));
iLenghtOfCompleteString:=len(sRawString);
iLenghtofStartIdentifier:=len(concat(sDataElementSeparator,sStringStartIdentifier));

IF iTemp > 0 THEN
	IF iLenghtofStartIdentifier > 1 THEN
		sTempString:=right(sRawString,(iLenghtOfCompleteString-iTemp-(iLenghtofStartIdentifier-1)));
	ELSE
		sTempString:=right(sRawString,(iLenghtOfCompleteString-iTemp));
	END_IF
	iTempStringEnd:=find(sTempString,sStringEndIdentifier);
	IF iTempStringEnd > 0 THEN
		sCutString:=MID(sTempString,iTempStringEnd-1,1);
	ELSE
		sCutString:='';	
	END_IF
ELSE
	sCutString:='';
END_IF
          
END_FUNCTION_BLOCK
